FUNCTION_BLOCK AssemblyActuatorGripper EXTENDS ZEquipment.ActuatorDigitalMonoPlusLsNo

METHOD PUBLIC AufAsync
VAR_INPUT
  startToken : ZCore.IStartToken;
END_VAR
MovePlusAsync(startToken:=startToken);
END_METHOD

METHOD PUBLIC Geschlossen : BOOL
VAR_INPUT
END_VAR
Geschlossen := IsAtMinus();
END_METHOD

METHOD PUBLIC Offen : BOOL
VAR_INPUT
END_VAR
Offen := IsAtPlus();
END_METHOD

METHOD PUBLIC ZuAsync
VAR_INPUT
  startToken : ZCore.IStartToken;
END_VAR
MoveMinusAsync(startToken:=startToken);
END_METHOD

END_FUNCTION_BLOCK

(* stored: Version 1.1.0.1
   POU AssemblyActuatorGripper: Id {49de3c57-0e79-426d-a9f7-08658d1e6ba8}, SpecialFunc None
   Method AufAsync: Id {d9b3fba8-ec46-4082-9cb7-f53a097a7164}
   Method Geschlossen: Id {ae0689b8-8156-4792-8380-557acc6754ae}
   Method Offen: Id {36aa3784-e3f8-4a16-ade3-d7c69fa4d96a}
   Method ZuAsync: Id {2abf578d-9146-4d98-ab85-e8cbf7282791} *)
